{attribute addProperty BoxType "EP9128-0021-0018"}
{attribute addProperty Id "A_0013_EP9128_0021_0019A_0013_EP9128_0021_0019_E94C525C4632579A_0010_EP9128_0021_0018_2_EP9128_1021EP9128_179A0949162A_0010_EP9128_0021_0018_3_EP9128_2021EP9128_179A0949162"}
{attribute addProperty CRC "2955987428"}
{attribute addProperty SizeInBites "4664"}
{attribute addProperty SizeInBytes "583"}
TYPE A_0010_EP9128_0021_0018_B030C9E4 EXTENDS EP9128_179A0949 :
STRUCT
	{attribute addProperty Name "A_0013_EP9128_0021_0019"}
	A_0013_EP9128_0021_0019 : A_0013_EP9128_0021_0019_E94C525C;
	{attribute addProperty Name "A_0010_EP9128_0021_0018_2_EP9128_1021"}
	A_0010_EP9128_0021_0018_2_EP9128_1021 : EP9128_179A0949;
	{attribute addProperty Name "A_0010_EP9128_0021_0018_3_EP9128_2021"}
	A_0010_EP9128_0021_0018_3_EP9128_2021 : EP9128_179A0949;
END_STRUCT
END_TYPE

(* stored: Version 1.2.0.0, ProductVersion 3.1.4024.9
   DUT A_0010_EP9128_0021_0018_B030C9E4: Id {edf69daf-2d94-4395-870a-ab48dd299944} *)
